{attribute 'qualified_only'}
{attribute 'strict'}
TYPE E_LoggerState :
(
	Open,
	Opening,
	Opening_Error,
	Opened,
	
	Writing,
	Writing_Error,
	
	Close,
	Closing,
	Closed,
	Closing_Error
) BYTE;
END_TYPE

(* stored: Version 1.1.0.1, ProductVersion 3.1.4024.11
   DUT E_LoggerState: Id {2e4f045d-024d-4b02-8f2e-df42c47bec90} *)
